RoboDK station: ME5286_Lab4_Serdoncillo_JustineJohnv2.rdk

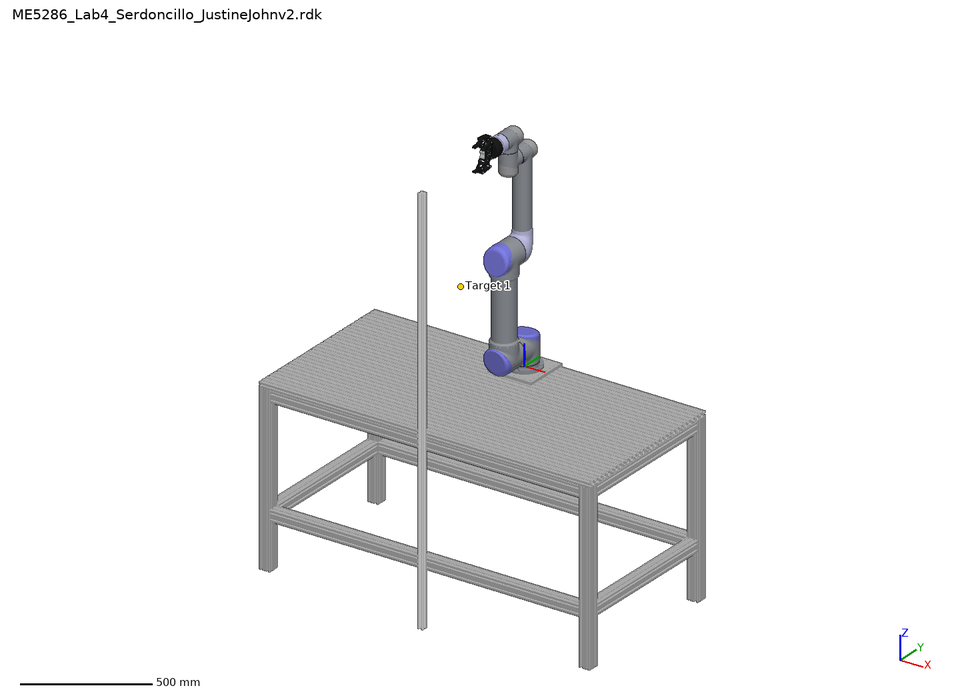
[picture v0: the station drawn from its stored meshes, robots at their saved joint values, targets as dots, program paths as lines]
Station ME5286_Lab4_Serdoncillo_JustineJohnv2 (saved by RoboDK 5.5.3). Poses are relative to the parent item; angles as X-Y-Z fixed-axis rotations.
  - frame UR5 Base at (0, 0, 0) mm
    - robot UR5: 6 axes, payload 5 kg, reach 850 mm, repeatability 0.1 mm, weight 18.4 kg
        modified DH rows (alpha deg, a mm, theta deg, d mm): 0, 0, 0, 89.2; 90, 0, 180, 0; 0, 425, 0, 0; 0, 392.43, 0, 109; -90, 0, 0, 93.65; 90, 0, 180, 82
        joint limits [-360, -360, -360, -360, -360, -360] to [360, 360, 360, 360, 360, 360]; home [0, -90, 90, 0, 90, 0]; saved at [0, -90, 0, -90, 0, 0]
      - tool Gripper RobotiQ 85 Opened, TCP at (0, 0, 149.6) mm, size 147.4 x 146.8 x 75 mm
    - target Target 1 (Cartesian target) at (-321.33, 39.91, 227.98) mm, rotated rx -179.55 ry -0.25 rz 179.77 deg; joints [-27.14, -115.32, 117.34, -92.04, -89.49, -206.91] of UR5
    - target Target 2 (Cartesian target) at (-321.33, 39.91, 227.98) mm, rotated rx -179.51 ry 0.14 rz 134.77 deg; joints [-27.14, -115.32, 117.34, -92.04, -89.49, -161.91] of UR5
    - target Target 3 (Cartesian target) at (-321.33, 39.91, 227.98) mm, rotated rx -179.51 ry 0.14 rz 134.77 deg; joints [-27.14, -115.32, 117.34, -92.04, -89.49, -86.91] of UR5
  - object table_base_setup at (0, 0, 0) mm, rotated rx 0 ry 0 rz -90 deg, size 1524 x 762 x 800.1 mm, geometry from table_base_setup.STEP
  - object 6ft_beam_table at (0, -675, 1000) mm, size 25.4 x 25.4 x 1828.8 mm, geometry from 6ft_beam_table.IGS
